{attribute addProperty BoxType "KL2012"}
{attribute addProperty Id "OutputAT %Q*BOOL000"}
{attribute addProperty CRC "3881556014"}
{attribute addProperty SizeInBites "0"}
{attribute addProperty SizeInBytes "0"}
TYPE Channel_E75BD82E :
STRUCT
	{attribute addProperty Name "Output"}
	Output AT %Q* : BOOL;
END_STRUCT
END_TYPE

(* stored: Version 1.2.0.0, ProductVersion 3.1.4024.9
   DUT Channel_E75BD82E: Id {a5ca78eb-c6e6-4a63-8fc3-01d0f69efe18} *)
